TYPE (* A Structured Data Type *)
  (* Standard: 61499-2 *)
  (* Version 0.9, 2012-01-10, IH, 4DIAC *)
  (* Compiler header: package fb.rt.test; *)
  (* ASN.1 tag APPLICATION 1 *)
  TestStruct : STRUCT
    FOO : BOOL;
    BAR : INT;
  END_STRUCT;
END_TYPE
